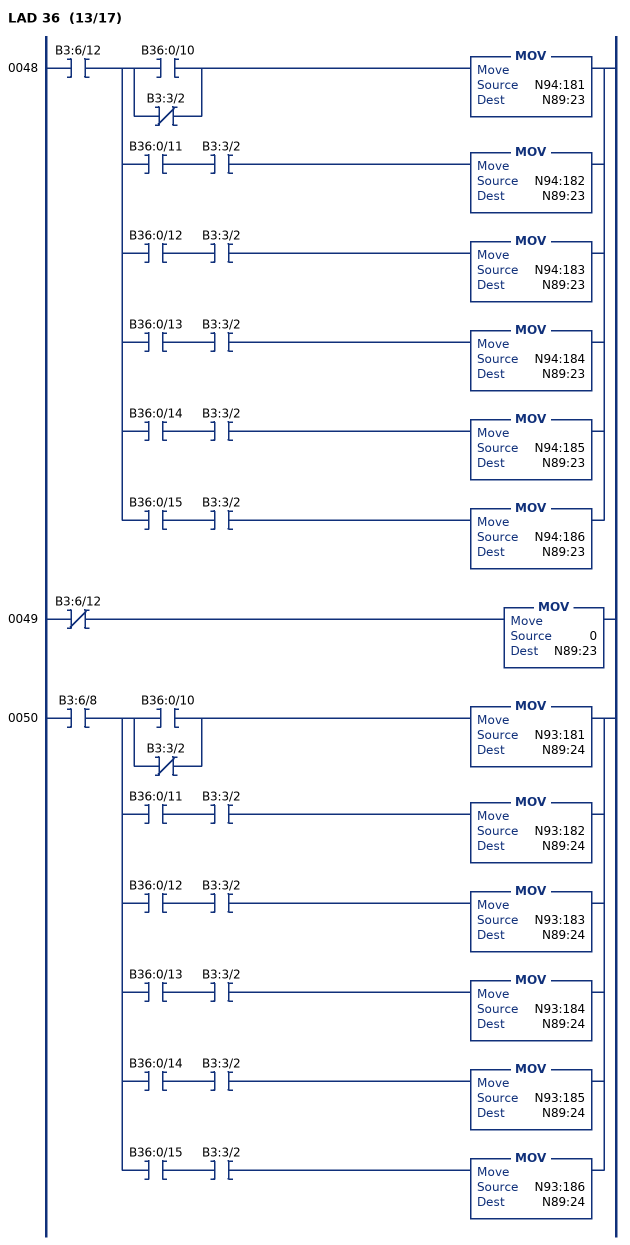
% Rung: 48 %
SOR XIC B3:6/12 BST BST XIC B36:0/10 NXB XIO B3:3/2 BND MOV N94:181 N89:23 NXB XIC B36:0/11 XIC B3:3/2 MOV N94:182 N89:23 NXB XIC B36:0/12 XIC B3:3/2 MOV N94:183 N89:23 NXB XIC B36:0/13 XIC B3:3/2 MOV N94:184 N89:23 NXB XIC B36:0/14 XIC B3:3/2 MOV N94:185 N89:23 NXB XIC B36:0/15 XIC B3:3/2 MOV N94:186 N89:23 BND EOR
% Rung: 49 %
SOR XIO B3:6/12 MOV 0 N89:23 EOR
% Rung: 50 %
SOR XIC B3:6/8 BST BST XIC B36:0/10 NXB XIO B3:3/2 BND MOV N93:181 N89:24 NXB XIC B36:0/11 XIC B3:3/2 MOV N93:182 N89:24 NXB XIC B36:0/12 XIC B3:3/2 MOV N93:183 N89:24 NXB XIC B36:0/13 XIC B3:3/2 MOV N93:184 N89:24 NXB XIC B36:0/14 XIC B3:3/2 MOV N93:185 N89:24 NXB XIC B36:0/15 XIC B3:3/2 MOV N93:186 N89:24 BND EOR

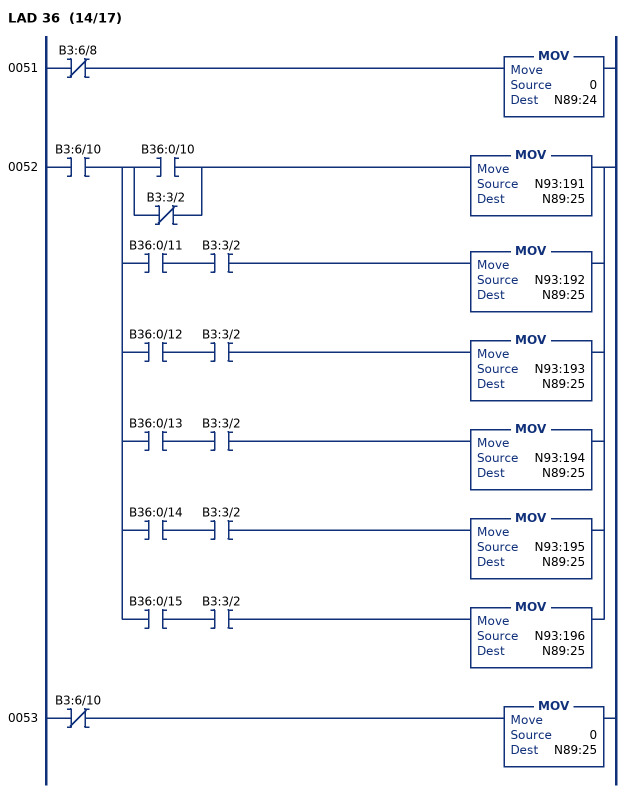
% Rung: 51 %
SOR XIO B3:6/8 MOV 0 N89:24 EOR
% Rung: 52 %
SOR XIC B3:6/10 BST BST XIC B36:0/10 NXB XIO B3:3/2 BND MOV N93:191 N89:25 NXB XIC B36:0/11 XIC B3:3/2 MOV N93:192 N89:25 NXB XIC B36:0/12 XIC B3:3/2 MOV N93:193 N89:25 NXB XIC B36:0/13 XIC B3:3/2 MOV N93:194 N89:25 NXB XIC B36:0/14 XIC B3:3/2 MOV N93:195 N89:25 NXB XIC B36:0/15 XIC B3:3/2 MOV N93:196 N89:25 BND EOR
% Rung: 53 %
SOR XIO B3:6/10 MOV 0 N89:25 EOR

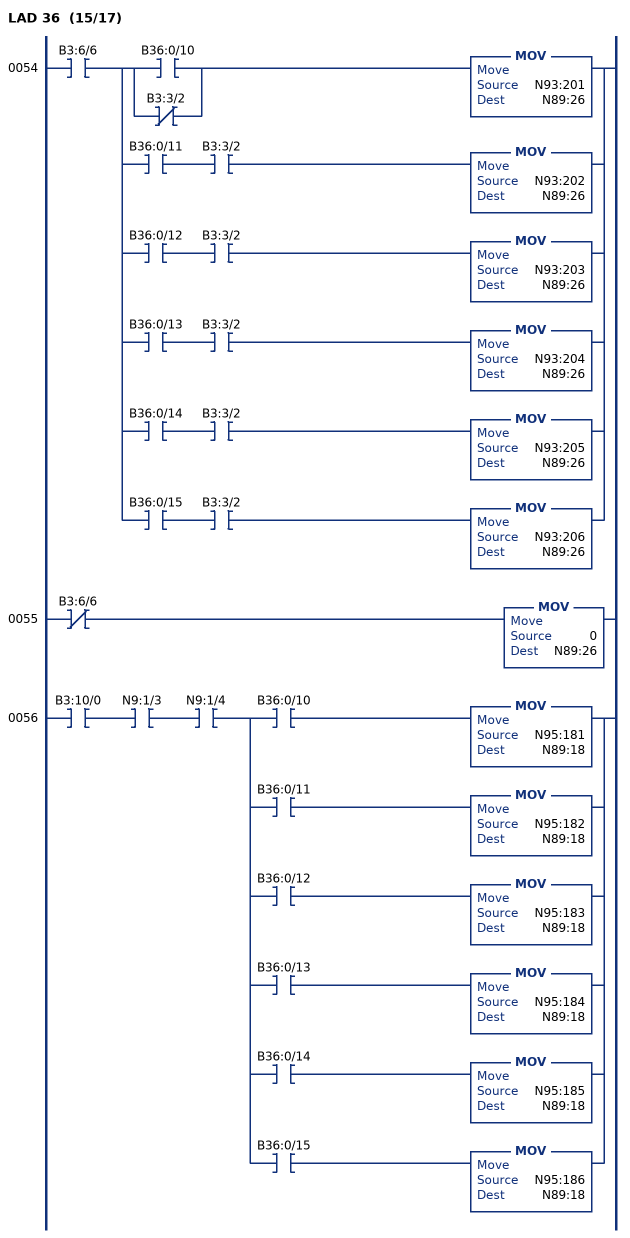
% Rung: 54 %
SOR XIC B3:6/6 BST BST XIC B36:0/10 NXB XIO B3:3/2 BND MOV N93:201 N89:26 NXB XIC B36:0/11 XIC B3:3/2 MOV N93:202 N89:26 NXB XIC B36:0/12 XIC B3:3/2 MOV N93:203 N89:26 NXB XIC B36:0/13 XIC B3:3/2 MOV N93:204 N89:26 NXB XIC B36:0/14 XIC B3:3/2 MOV N93:205 N89:26 NXB XIC B36:0/15 XIC B3:3/2 MOV N93:206 N89:26 BND EOR
% Rung: 55 %
SOR XIO B3:6/6 MOV 0 N89:26 EOR
% Rung: 56 %
SOR XIC B3:10/0 XIC N9:1/3 XIC N9:1/4 BST XIC B36:0/10 MOV N95:181 N89:18 NXB XIC B36:0/11 MOV N95:182 N89:18 NXB XIC B36:0/12 MOV N95:183 N89:18 NXB XIC B36:0/13 MOV N95:184 N89:18 NXB XIC B36:0/14 MOV N95:185 N89:18 NXB XIC B36:0/15 MOV N95:186 N89:18 BND EOR

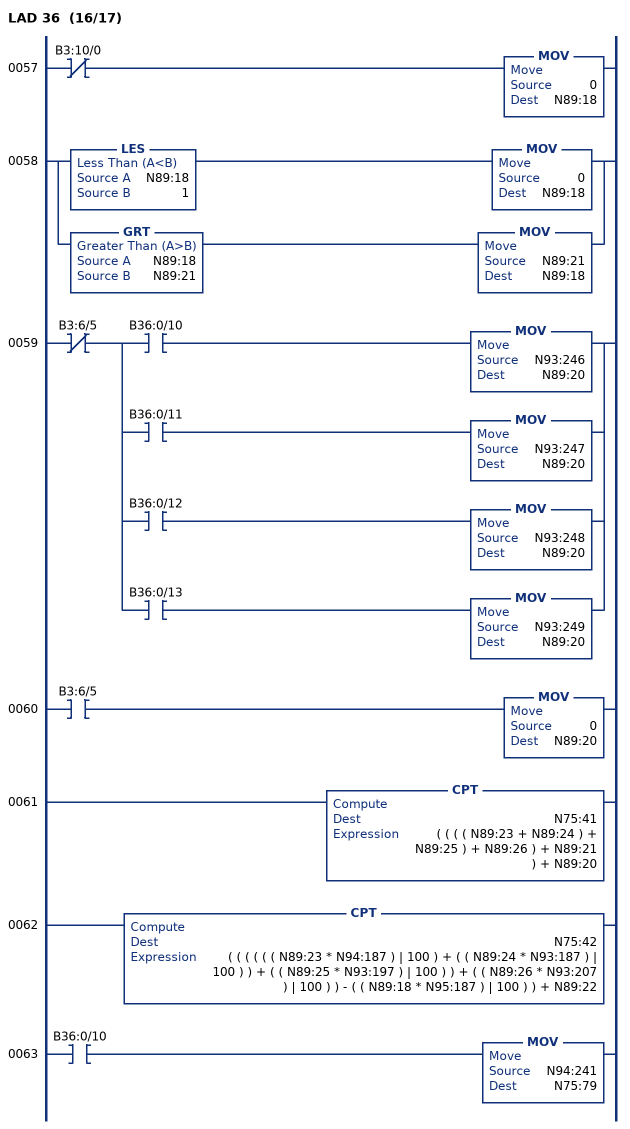
% Rung: 57 %
SOR XIO B3:10/0 MOV 0 N89:18 EOR
% Rung: 58 %
SOR BST LES N89:18 1 MOV 0 N89:18 NXB GRT N89:18 N89:21 MOV N89:21 N89:18 BND EOR
% Rung: 59 %
SOR XIO B3:6/5 BST XIC B36:0/10 MOV N93:246 N89:20 NXB XIC B36:0/11 MOV N93:247 N89:20 NXB XIC B36:0/12 MOV N93:248 N89:20 NXB XIC B36:0/13 MOV N93:249 N89:20 BND EOR
% Rung: 60 %
SOR XIC B3:6/5 MOV 0 N89:20 EOR
% Rung: 61 %
SOR CPT N75:41 " ( ( ( ( N89:23 + N89:24 ) + N89:25 ) + N89:26 ) + N89:21 ) + N89:20 " EOR
% Rung: 62 %
SOR CPT N75:42 " ( ( ( ( ( ( N89:23 * N94:187 ) | 100 ) + ( ( N89:24 * N93:187 ) | 100 ) ) + ( ( N89:25 * N93:197 ) | 100 ) ) + ( ( N89:26 * N93:207 ) | 100 ) ) - ( ( N89:18 * N95:187 ) | 100 ) ) + N89:22 " EOR
% Rung: 63 %
SOR XIC B36:0/10 MOV N94:241 N75:79 EOR

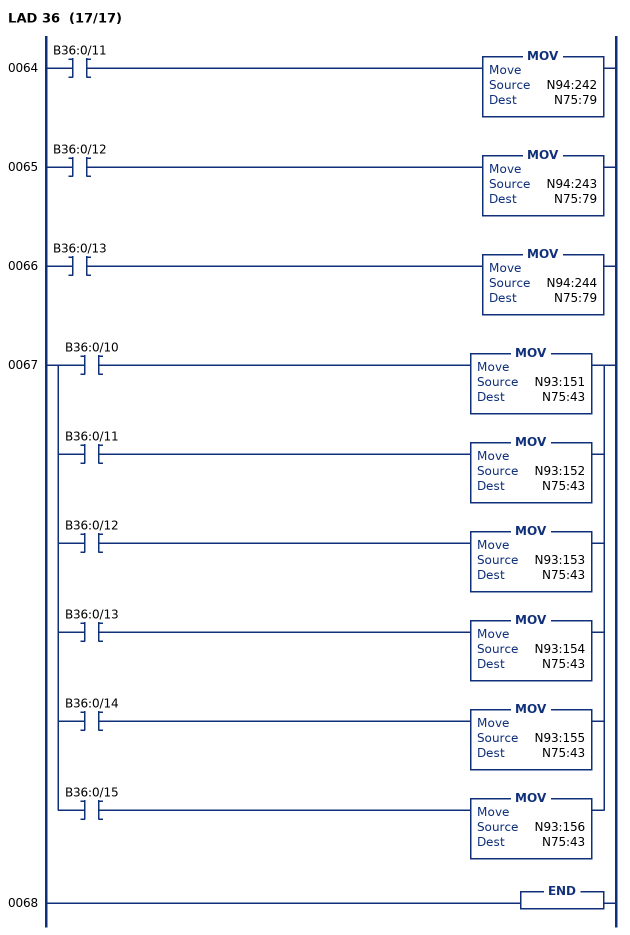
% Rung: 64 %
SOR XIC B36:0/11 MOV N94:242 N75:79 EOR
% Rung: 65 %
SOR XIC B36:0/12 MOV N94:243 N75:79 EOR
% Rung: 66 %
SOR XIC B36:0/13 MOV N94:244 N75:79 EOR
% Rung: 67 %
SOR BST XIC B36:0/10 MOV N93:151 N75:43 NXB XIC B36:0/11 MOV N93:152 N75:43 NXB XIC B36:0/12 MOV N93:153 N75:43 NXB XIC B36:0/13 MOV N93:154 N75:43 NXB XIC B36:0/14 MOV N93:155 N75:43 NXB XIC B36:0/15 MOV N93:156 N75:43 BND EOR
% Rung: 68 %
SOR END EOR

LADDER 41
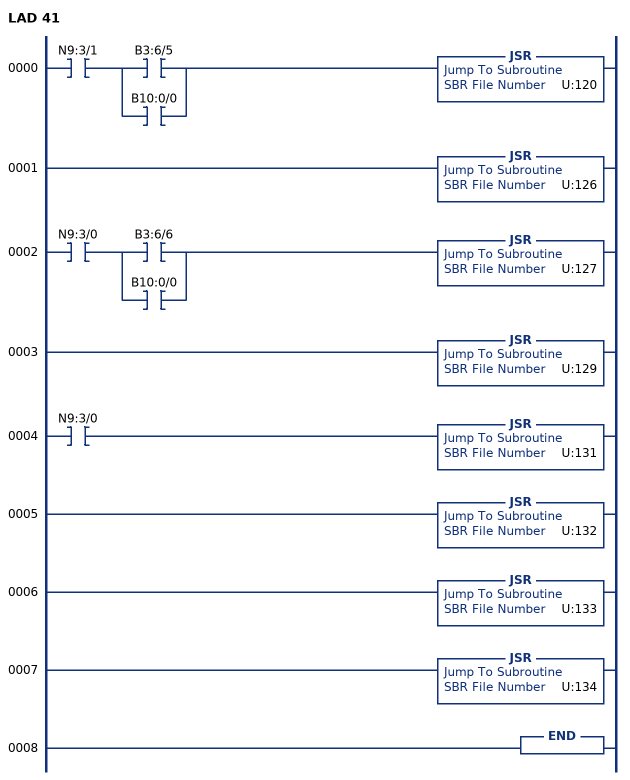
% Rung: 0 %
SOR XIC N9:3/1 BST XIC B3:6/5 NXB XIC B10:0/0 BND JSR U:120 EOR
% Rung: 1 %
SOR JSR U:126 EOR
% Rung: 2 %
SOR XIC N9:3/0 BST XIC B3:6/6 NXB XIC B10:0/0 BND JSR U:127 EOR
% Rung: 3 %
SOR JSR U:129 EOR
% Rung: 4 %
SOR XIC N9:3/0 JSR U:131 EOR
% Rung: 5 %
SOR JSR U:132 EOR
% Rung: 6 %
SOR JSR U:133 EOR
% Rung: 7 %
SOR JSR U:134 EOR
% Rung: 8 %
SOR END EOR

LADDER 50
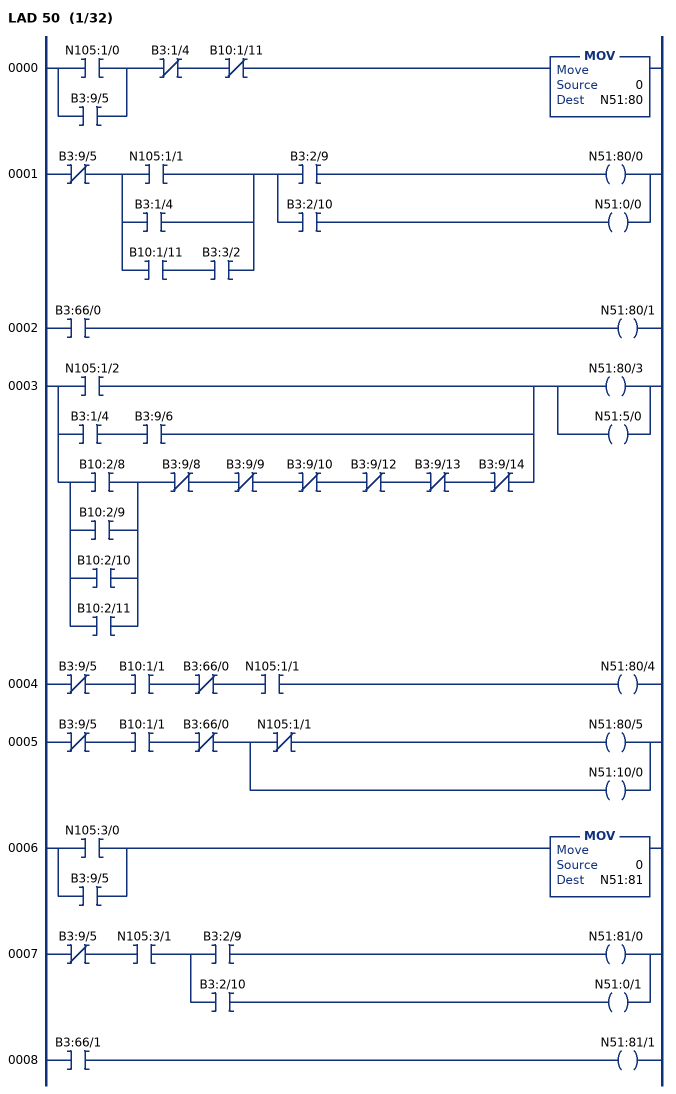
% Rung: 0 %
SOR BST XIC N105:1/0 NXB XIC B3:9/5 BND XIO B3:1/4 XIO B10:1/11 MOV 0 N51:80 EOR
% Rung: 1 %
SOR XIO B3:9/5 BST XIC N105:1/1 NXB XIC B3:1/4 NXB XIC B10:1/11 XIC B3:3/2 BND BST XIC B3:2/9 OTE N51:80/0 NXB XIC B3:2/10 OTE N51:0/0 BND EOR
% Rung: 2 %
SOR XIC B3:66/0 OTE N51:80/1 EOR
% Rung: 3 %
SOR BST XIC N105:1/2 NXB XIC B3:1/4 XIC B3:9/6 NXB BST XIC B10:2/8 NXB XIC B10:2/9 NXB XIC B10:2/10 NXB XIC B10:2/11 BND XIO B3:9/8 XIO B3:9/9 XIO B3:9/10 XIO B3:9/12 XIO B3:9/13 XIO B3:9/14 BND BST OTE N51:80/3 NXB OTE N51:5/0 BND EOR
% Rung: 4 %
SOR XIO B3:9/5 XIC B10:1/1 XIO B3:66/0 XIC N105:1/1 OTE N51:80/4 EOR
% Rung: 5 %
SOR XIO B3:9/5 XIC B10:1/1 XIO B3:66/0 BST XIO N105:1/1 OTE N51:80/5 NXB OTE N51:10/0 BND EOR
% Rung: 6 %
SOR BST XIC N105:3/0 NXB XIC B3:9/5 BND MOV 0 N51:81 EOR
% Rung: 7 %
SOR XIO B3:9/5 XIC N105:3/1 BST XIC B3:2/9 OTE N51:81/0 NXB XIC B3:2/10 OTE N51:0/1 BND EOR
% Rung: 8 %
SOR XIC B3:66/1 OTE N51:81/1 EOR

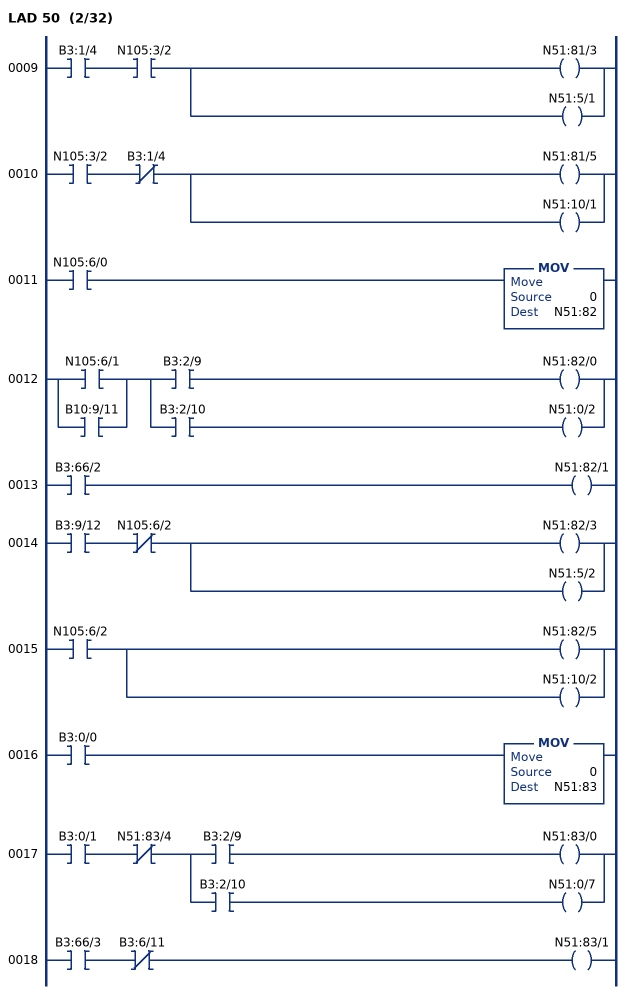
% Rung: 9 %
SOR XIC B3:1/4 XIC N105:3/2 BST OTE N51:81/3 NXB OTE N51:5/1 BND EOR
% Rung: 10 %
SOR XIC N105:3/2 XIO B3:1/4 BST OTE N51:81/5 NXB OTE N51:10/1 BND EOR
% Rung: 11 %
SOR XIC N105:6/0 MOV 0 N51:82 EOR
% Rung: 12 %
SOR BST XIC N105:6/1 NXB XIC B10:9/11 BND BST XIC B3:2/9 OTE N51:82/0 NXB XIC B3:2/10 OTE N51:0/2 BND EOR
% Rung: 13 %
SOR XIC B3:66/2 OTE N51:82/1 EOR
% Rung: 14 %
SOR XIC B3:9/12 XIO N105:6/2 BST OTE N51:82/3 NXB OTE N51:5/2 BND EOR
% Rung: 15 %
SOR XIC N105:6/2 BST OTE N51:82/5 NXB OTE N51:10/2 BND EOR
% Rung: 16 %
SOR XIC B3:0/0 MOV 0 N51:83 EOR
% Rung: 17 %
SOR XIC B3:0/1 XIO N51:83/4 BST XIC B3:2/9 OTE N51:83/0 NXB XIC B3:2/10 OTE N51:0/7 BND EOR
% Rung: 18 %
SOR XIC B3:66/3 XIO B3:6/11 OTE N51:83/1 EOR

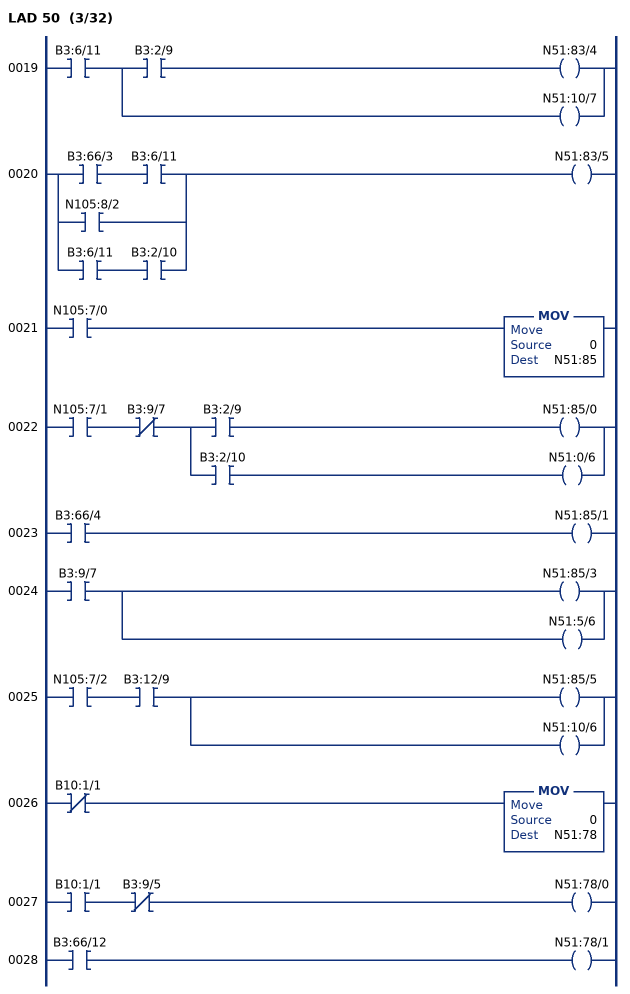
% Rung: 19 %
SOR XIC B3:6/11 BST XIC B3:2/9 OTE N51:83/4 NXB OTE N51:10/7 BND EOR
% Rung: 20 %
SOR BST XIC B3:66/3 XIC B3:6/11 NXB XIC N105:8/2 NXB XIC B3:6/11 XIC B3:2/10 BND OTE N51:83/5 EOR
% Rung: 21 %
SOR XIC N105:7/0 MOV 0 N51:85 EOR
% Rung: 22 %
SOR XIC N105:7/1 XIO B3:9/7 BST XIC B3:2/9 OTE N51:85/0 NXB XIC B3:2/10 OTE N51:0/6 BND EOR
% Rung: 23 %
SOR XIC B3:66/4 OTE N51:85/1 EOR
% Rung: 24 %
SOR XIC B3:9/7 BST OTE N51:85/3 NXB OTE N51:5/6 BND EOR
% Rung: 25 %
SOR XIC N105:7/2 XIC B3:12/9 BST OTE N51:85/5 NXB OTE N51:10/6 BND EOR
% Rung: 26 %
SOR XIO B10:1/1 MOV 0 N51:78 EOR
% Rung: 27 %
SOR XIC B10:1/1 XIO B3:9/5 OTE N51:78/0 EOR
% Rung: 28 %
SOR XIC B3:66/12 OTE N51:78/1 EOR

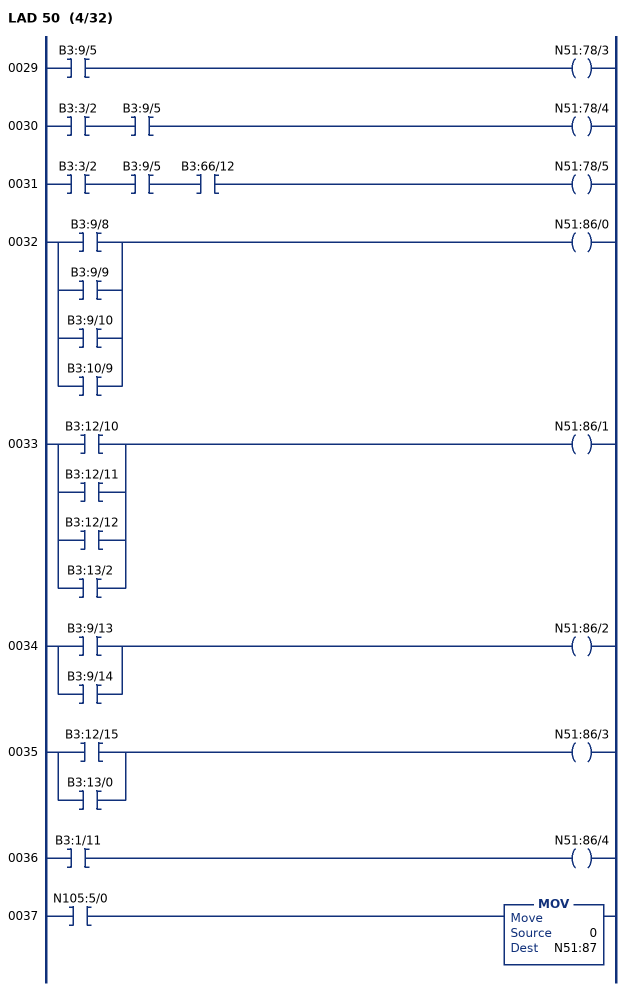
% Rung: 29 %
SOR XIC B3:9/5 OTE N51:78/3 EOR
% Rung: 30 %
SOR XIC B3:3/2 XIC B3:9/5 OTE N51:78/4 EOR
% Rung: 31 %
SOR XIC B3:3/2 XIC B3:9/5 XIC B3:66/12 OTE N51:78/5 EOR
% Rung: 32 %
SOR BST XIC B3:9/8 NXB XIC B3:9/9 NXB XIC B3:9/10 NXB XIC B3:10/9 BND OTE N51:86/0 EOR
% Rung: 33 %
SOR BST XIC B3:12/10 NXB XIC B3:12/11 NXB XIC B3:12/12 NXB XIC B3:13/2 BND OTE N51:86/1 EOR
% Rung: 34 %
SOR BST XIC B3:9/13 NXB XIC B3:9/14 BND OTE N51:86/2 EOR
% Rung: 35 %
SOR BST XIC B3:12/15 NXB XIC B3:13/0 BND OTE N51:86/3 EOR
% Rung: 36 %
SOR XIC B3:1/11 OTE N51:86/4 EOR
% Rung: 37 %
SOR XIC N105:5/0 MOV 0 N51:87 EOR

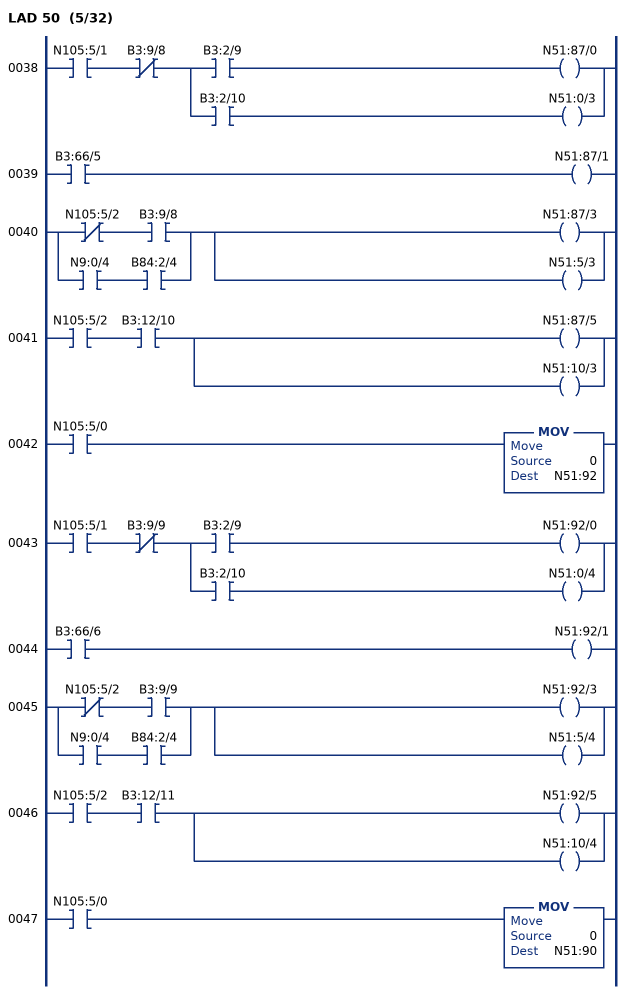
% Rung: 38 %
SOR XIC N105:5/1 XIO B3:9/8 BST XIC B3:2/9 OTE N51:87/0 NXB XIC B3:2/10 OTE N51:0/3 BND EOR
% Rung: 39 %
SOR XIC B3:66/5 OTE N51:87/1 EOR
% Rung: 40 %
SOR BST XIO N105:5/2 XIC B3:9/8 NXB XIC N9:0/4 XIC B84:2/4 BND BST OTE N51:87/3 NXB OTE N51:5/3 BND EOR
% Rung: 41 %
SOR XIC N105:5/2 XIC B3:12/10 BST OTE N51:87/5 NXB OTE N51:10/3 BND EOR
% Rung: 42 %
SOR XIC N105:5/0 MOV 0 N51:92 EOR
% Rung: 43 %
SOR XIC N105:5/1 XIO B3:9/9 BST XIC B3:2/9 OTE N51:92/0 NXB XIC B3:2/10 OTE N51:0/4 BND EOR
% Rung: 44 %
SOR XIC B3:66/6 OTE N51:92/1 EOR
% Rung: 45 %
SOR BST XIO N105:5/2 XIC B3:9/9 NXB XIC N9:0/4 XIC B84:2/4 BND BST OTE N51:92/3 NXB OTE N51:5/4 BND EOR
% Rung: 46 %
SOR XIC N105:5/2 XIC B3:12/11 BST OTE N51:92/5 NXB OTE N51:10/4 BND EOR
% Rung: 47 %
SOR XIC N105:5/0 MOV 0 N51:90 EOR

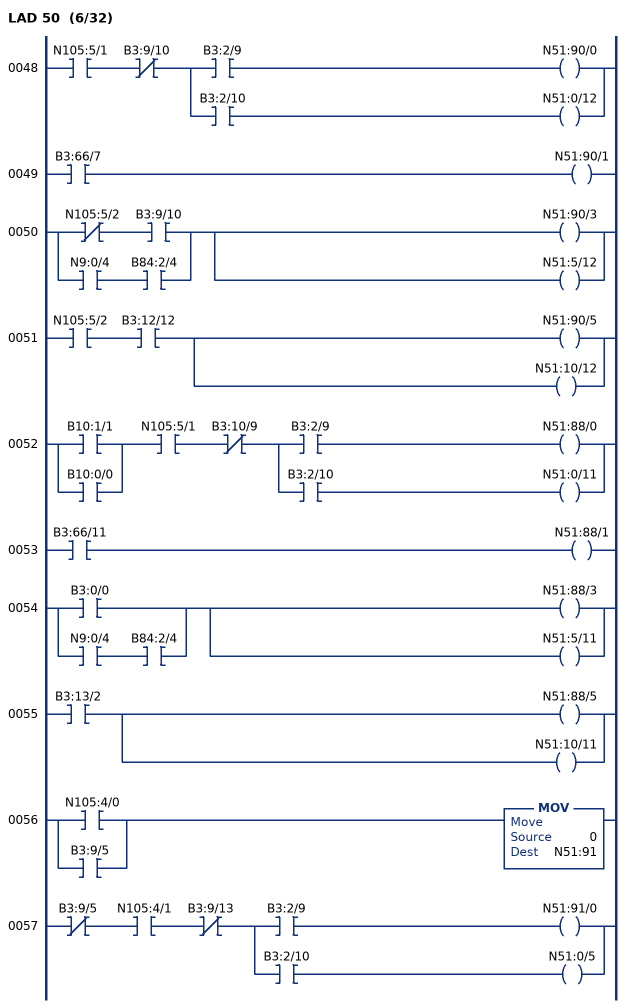
% Rung: 48 %
SOR XIC N105:5/1 XIO B3:9/10 BST XIC B3:2/9 OTE N51:90/0 NXB XIC B3:2/10 OTE N51:0/12 BND EOR
% Rung: 49 %
SOR XIC B3:66/7 OTE N51:90/1 EOR
% Rung: 50 %
SOR BST XIO N105:5/2 XIC B3:9/10 NXB XIC N9:0/4 XIC B84:2/4 BND BST OTE N51:90/3 NXB OTE N51:5/12 BND EOR
% Rung: 51 %
SOR XIC N105:5/2 XIC B3:12/12 BST OTE N51:90/5 NXB OTE N51:10/12 BND EOR
% Rung: 52 %
SOR BST XIC B10:1/1 NXB XIC B10:0/0 BND XIC N105:5/1 XIO B3:10/9 BST XIC B3:2/9 OTE N51:88/0 NXB XIC B3:2/10 OTE N51:0/11 BND EOR
% Rung: 53 %
SOR XIC B3:66/11 OTE N51:88/1 EOR
% Rung: 54 %
SOR BST XIC B3:0/0 NXB XIC N9:0/4 XIC B84:2/4 BND BST OTE N51:88/3 NXB OTE N51:5/11 BND EOR
% Rung: 55 %
SOR XIC B3:13/2 BST OTE N51:88/5 NXB OTE N51:10/11 BND EOR
% Rung: 56 %
SOR BST XIC N105:4/0 NXB XIC B3:9/5 BND MOV 0 N51:91 EOR
% Rung: 57 %
SOR XIO B3:9/5 XIC N105:4/1 XIO B3:9/13 BST XIC B3:2/9 OTE N51:91/0 NXB XIC B3:2/10 OTE N51:0/5 BND EOR

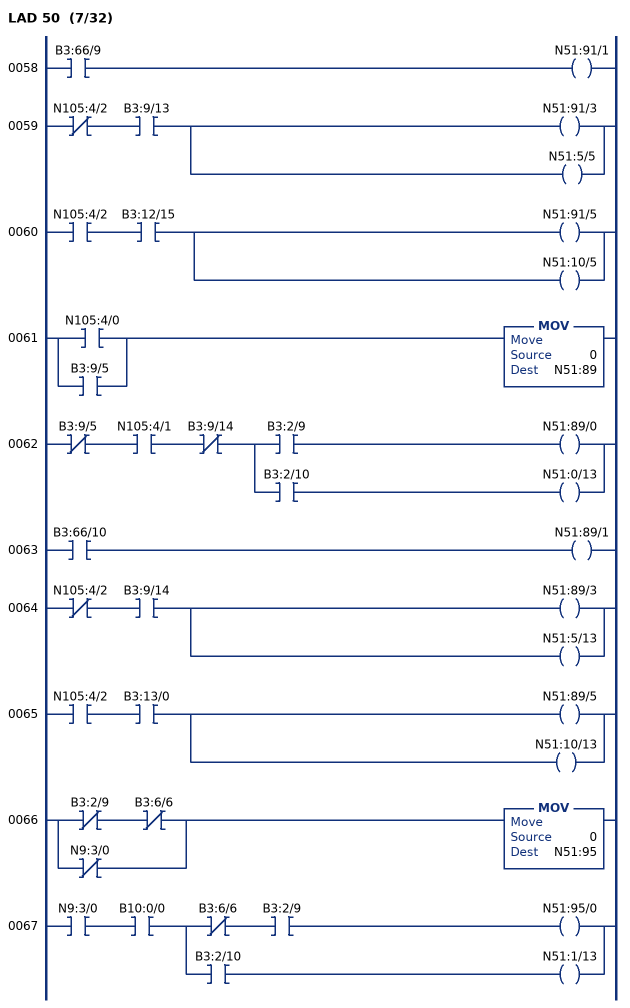
% Rung: 58 %
SOR XIC B3:66/9 OTE N51:91/1 EOR
% Rung: 59 %
SOR XIO N105:4/2 XIC B3:9/13 BST OTE N51:91/3 NXB OTE N51:5/5 BND EOR
% Rung: 60 %
SOR XIC N105:4/2 XIC B3:12/15 BST OTE N51:91/5 NXB OTE N51:10/5 BND EOR
% Rung: 61 %
SOR BST XIC N105:4/0 NXB XIC B3:9/5 BND MOV 0 N51:89 EOR
% Rung: 62 %
SOR XIO B3:9/5 XIC N105:4/1 XIO B3:9/14 BST XIC B3:2/9 OTE N51:89/0 NXB XIC B3:2/10 OTE N51:0/13 BND EOR
% Rung: 63 %
SOR XIC B3:66/10 OTE N51:89/1 EOR
% Rung: 64 %
SOR XIO N105:4/2 XIC B3:9/14 BST OTE N51:89/3 NXB OTE N51:5/13 BND EOR
% Rung: 65 %
SOR XIC N105:4/2 XIC B3:13/0 BST OTE N51:89/5 NXB OTE N51:10/13 BND EOR
% Rung: 66 %
SOR BST XIO B3:2/9 XIO B3:6/6 NXB XIO N9:3/0 BND MOV 0 N51:95 EOR
% Rung: 67 %
SOR XIC N9:3/0 XIC B10:0/0 BST XIO B3:6/6 XIC B3:2/9 OTE N51:95/0 NXB XIC B3:2/10 OTE N51:1/13 BND EOR

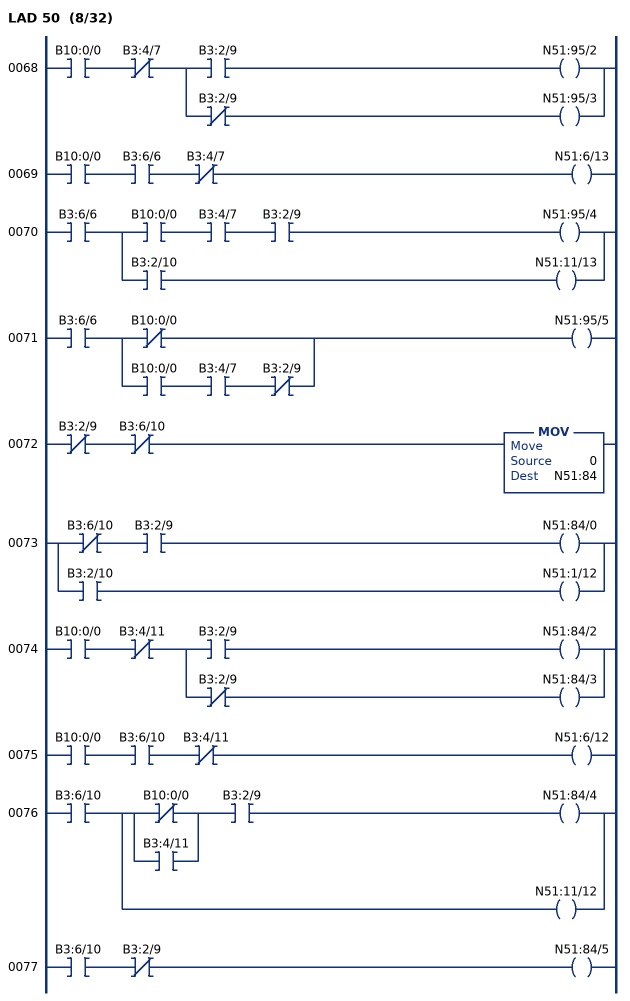
% Rung: 68 %
SOR XIC B10:0/0 XIO B3:4/7 BST XIC B3:2/9 OTE N51:95/2 NXB XIO B3:2/9 OTE N51:95/3 BND EOR
% Rung: 69 %
SOR XIC B10:0/0 XIC B3:6/6 XIO B3:4/7 OTE N51:6/13 EOR
% Rung: 70 %
SOR XIC B3:6/6 BST XIC B10:0/0 XIC B3:4/7 XIC B3:2/9 OTE N51:95/4 NXB XIC B3:2/10 OTE N51:11/13 BND EOR
% Rung: 71 %
SOR XIC B3:6/6 BST XIO B10:0/0 NXB XIC B10:0/0 XIC B3:4/7 XIO B3:2/9 BND OTE N51:95/5 EOR
% Rung: 72 %
SOR XIO B3:2/9 XIO B3:6/10 MOV 0 N51:84 EOR
% Rung: 73 %
SOR BST XIO B3:6/10 XIC B3:2/9 OTE N51:84/0 NXB XIC B3:2/10 OTE N51:1/12 BND EOR
% Rung: 74 %
SOR XIC B10:0/0 XIO B3:4/11 BST XIC B3:2/9 OTE N51:84/2 NXB XIO B3:2/9 OTE N51:84/3 BND EOR
% Rung: 75 %
SOR XIC B10:0/0 XIC B3:6/10 XIO B3:4/11 OTE N51:6/12 EOR
% Rung: 76 %
SOR XIC B3:6/10 BST BST XIO B10:0/0 NXB XIC B3:4/11 BND XIC B3:2/9 OTE N51:84/4 NXB OTE N51:11/12 BND EOR
% Rung: 77 %
SOR XIC B3:6/10 XIO B3:2/9 OTE N51:84/5 EOR

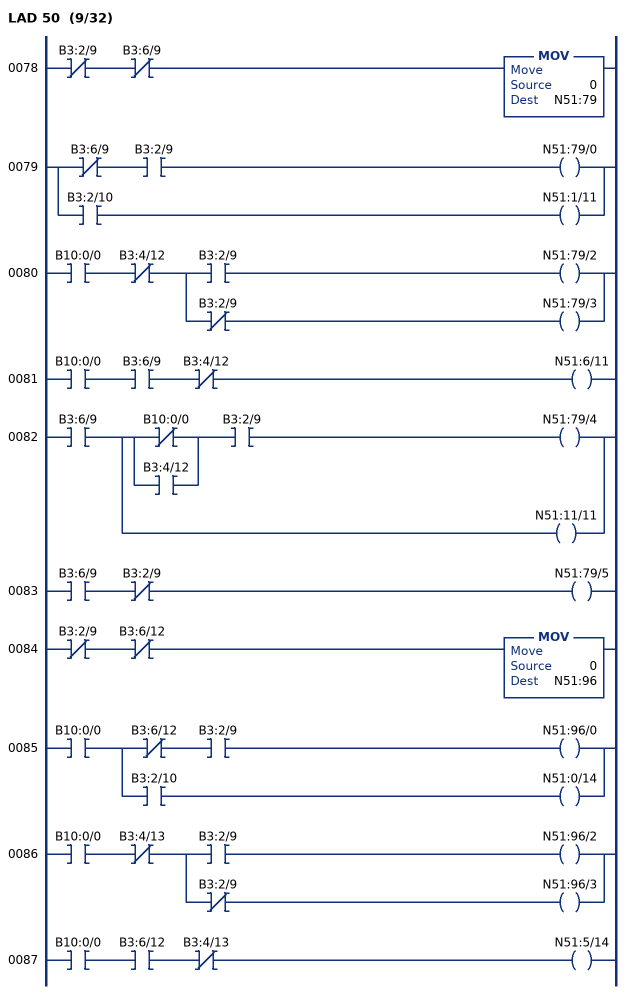
% Rung: 78 %
SOR XIO B3:2/9 XIO B3:6/9 MOV 0 N51:79 EOR
% Rung: 79 %
SOR BST XIO B3:6/9 XIC B3:2/9 OTE N51:79/0 NXB XIC B3:2/10 OTE N51:1/11 BND EOR
% Rung: 80 %
SOR XIC B10:0/0 XIO B3:4/12 BST XIC B3:2/9 OTE N51:79/2 NXB XIO B3:2/9 OTE N51:79/3 BND EOR
% Rung: 81 %
SOR XIC B10:0/0 XIC B3:6/9 XIO B3:4/12 OTE N51:6/11 EOR
% Rung: 82 %
SOR XIC B3:6/9 BST BST XIO B10:0/0 NXB XIC B3:4/12 BND XIC B3:2/9 OTE N51:79/4 NXB OTE N51:11/11 BND EOR
% Rung: 83 %
SOR XIC B3:6/9 XIO B3:2/9 OTE N51:79/5 EOR
% Rung: 84 %
SOR XIO B3:2/9 XIO B3:6/12 MOV 0 N51:96 EOR
% Rung: 85 %
SOR XIC B10:0/0 BST XIO B3:6/12 XIC B3:2/9 OTE N51:96/0 NXB XIC B3:2/10 OTE N51:0/14 BND EOR
% Rung: 86 %
SOR XIC B10:0/0 XIO B3:4/13 BST XIC B3:2/9 OTE N51:96/2 NXB XIO B3:2/9 OTE N51:96/3 BND EOR
% Rung: 87 %
SOR XIC B10:0/0 XIC B3:6/12 XIO B3:4/13 OTE N51:5/14 EOR

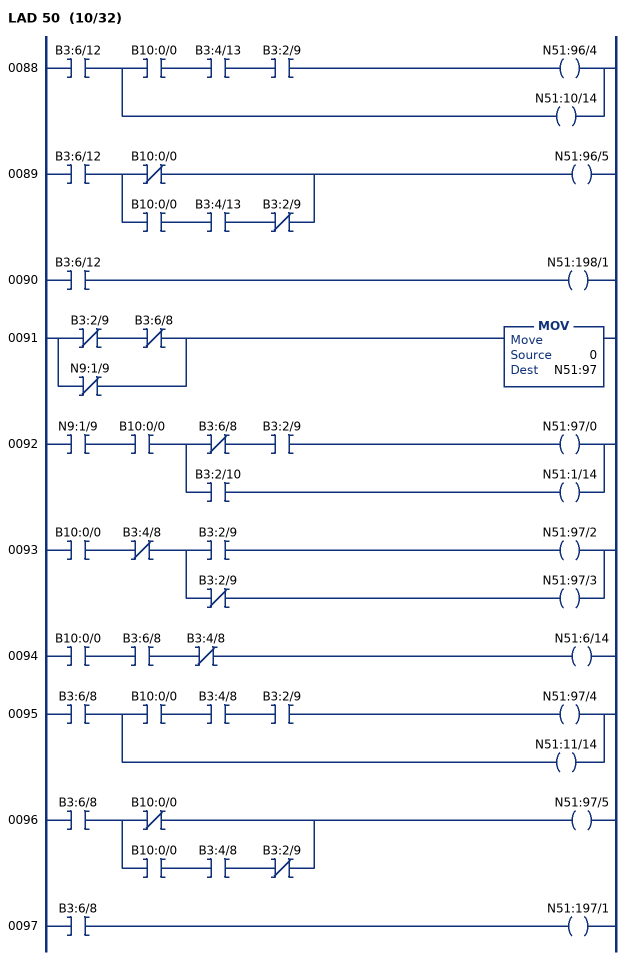
% Rung: 88 %
SOR XIC B3:6/12 BST XIC B10:0/0 XIC B3:4/13 XIC B3:2/9 OTE N51:96/4 NXB OTE N51:10/14 BND EOR
% Rung: 89 %
SOR XIC B3:6/12 BST XIO B10:0/0 NXB XIC B10:0/0 XIC B3:4/13 XIO B3:2/9 BND OTE N51:96/5 EOR
% Rung: 90 %
SOR XIC B3:6/12 OTE N51:198/1 EOR
% Rung: 91 %
SOR BST XIO B3:2/9 XIO B3:6/8 NXB XIO N9:1/9 BND MOV 0 N51:97 EOR
% Rung: 92 %
SOR XIC N9:1/9 XIC B10:0/0 BST XIO B3:6/8 XIC B3:2/9 OTE N51:97/0 NXB XIC B3:2/10 OTE N51:1/14 BND EOR
% Rung: 93 %
SOR XIC B10:0/0 XIO B3:4/8 BST XIC B3:2/9 OTE N51:97/2 NXB XIO B3:2/9 OTE N51:97/3 BND EOR
% Rung: 94 %
SOR XIC B10:0/0 XIC B3:6/8 XIO B3:4/8 OTE N51:6/14 EOR
% Rung: 95 %
SOR XIC B3:6/8 BST XIC B10:0/0 XIC B3:4/8 XIC B3:2/9 OTE N51:97/4 NXB OTE N51:11/14 BND EOR
% Rung: 96 %
SOR XIC B3:6/8 BST XIO B10:0/0 NXB XIC B10:0/0 XIC B3:4/8 XIO B3:2/9 BND OTE N51:97/5 EOR
% Rung: 97 %
SOR XIC B3:6/8 OTE N51:197/1 EOR

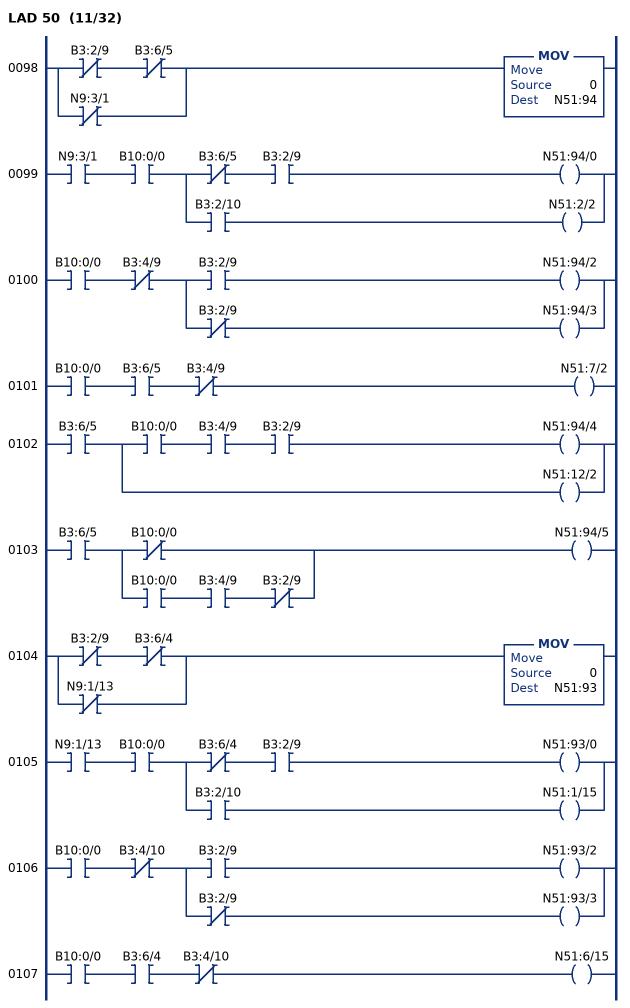
% Rung: 98 %
SOR BST XIO B3:2/9 XIO B3:6/5 NXB XIO N9:3/1 BND MOV 0 N51:94 EOR
% Rung: 99 %
SOR XIC N9:3/1 XIC B10:0/0 BST XIO B3:6/5 XIC B3:2/9 OTE N51:94/0 NXB XIC B3:2/10 OTE N51:2/2 BND EOR
% Rung: 100 %
SOR XIC B10:0/0 XIO B3:4/9 BST XIC B3:2/9 OTE N51:94/2 NXB XIO B3:2/9 OTE N51:94/3 BND EOR
% Rung: 101 %
SOR XIC B10:0/0 XIC B3:6/5 XIO B3:4/9 OTE N51:7/2 EOR
% Rung: 102 %
SOR XIC B3:6/5 BST XIC B10:0/0 XIC B3:4/9 XIC B3:2/9 OTE N51:94/4 NXB OTE N51:12/2 BND EOR
% Rung: 103 %
SOR XIC B3:6/5 BST XIO B10:0/0 NXB XIC B10:0/0 XIC B3:4/9 XIO B3:2/9 BND OTE N51:94/5 EOR
% Rung: 104 %
SOR BST XIO B3:2/9 XIO B3:6/4 NXB XIO N9:1/13 BND MOV 0 N51:93 EOR
% Rung: 105 %
SOR XIC N9:1/13 XIC B10:0/0 BST XIO B3:6/4 XIC B3:2/9 OTE N51:93/0 NXB XIC B3:2/10 OTE N51:1/15 BND EOR
% Rung: 106 %
SOR XIC B10:0/0 XIO B3:4/10 BST XIC B3:2/9 OTE N51:93/2 NXB XIO B3:2/9 OTE N51:93/3 BND EOR
% Rung: 107 %
SOR XIC B10:0/0 XIC B3:6/4 XIO B3:4/10 OTE N51:6/15 EOR

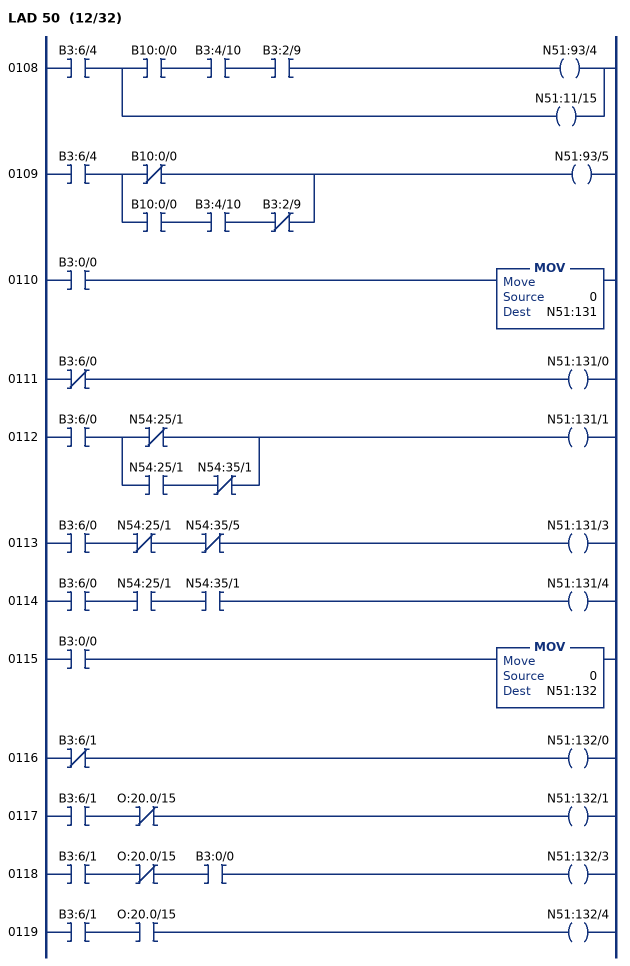
% Rung: 108 %
SOR XIC B3:6/4 BST XIC B10:0/0 XIC B3:4/10 XIC B3:2/9 OTE N51:93/4 NXB OTE N51:11/15 BND EOR
% Rung: 109 %
SOR XIC B3:6/4 BST XIO B10:0/0 NXB XIC B10:0/0 XIC B3:4/10 XIO B3:2/9 BND OTE N51:93/5 EOR
% Rung: 110 %
SOR XIC B3:0/0 MOV 0 N51:131 EOR
% Rung: 111 %
SOR XIO B3:6/0 OTE N51:131/0 EOR
% Rung: 112 %
SOR XIC B3:6/0 BST XIO N54:25/1 NXB XIC N54:25/1 XIO N54:35/1 BND OTE N51:131/1 EOR
% Rung: 113 %
SOR XIC B3:6/0 XIO N54:25/1 XIO N54:35/5 OTE N51:131/3 EOR
% Rung: 114 %
SOR XIC B3:6/0 XIC N54:25/1 XIC N54:35/1 OTE N51:131/4 EOR
% Rung: 115 %
SOR XIC B3:0/0 MOV 0 N51:132 EOR
% Rung: 116 %
SOR XIO B3:6/1 OTE N51:132/0 EOR
% Rung: 117 %
SOR XIC B3:6/1 XIO O:20.0/15 OTE N51:132/1 EOR
% Rung: 118 %
SOR XIC B3:6/1 XIO O:20.0/15 XIC B3:0/0 OTE N51:132/3 EOR
% Rung: 119 %
SOR XIC B3:6/1 XIC O:20.0/15 OTE N51:132/4 EOR

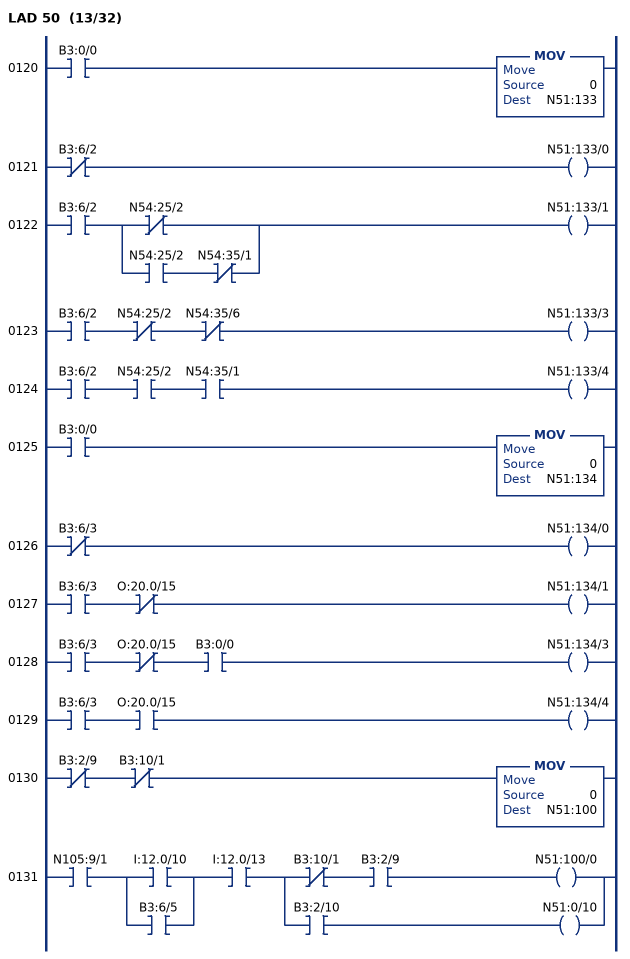
% Rung: 120 %
SOR XIC B3:0/0 MOV 0 N51:133 EOR
% Rung: 121 %
SOR XIO B3:6/2 OTE N51:133/0 EOR
% Rung: 122 %
SOR XIC B3:6/2 BST XIO N54:25/2 NXB XIC N54:25/2 XIO N54:35/1 BND OTE N51:133/1 EOR
% Rung: 123 %
SOR XIC B3:6/2 XIO N54:25/2 XIO N54:35/6 OTE N51:133/3 EOR
% Rung: 124 %
SOR XIC B3:6/2 XIC N54:25/2 XIC N54:35/1 OTE N51:133/4 EOR
% Rung: 125 %
SOR XIC B3:0/0 MOV 0 N51:134 EOR
% Rung: 126 %
SOR XIO B3:6/3 OTE N51:134/0 EOR
% Rung: 127 %
SOR XIC B3:6/3 XIO O:20.0/15 OTE N51:134/1 EOR
% Rung: 128 %
SOR XIC B3:6/3 XIO O:20.0/15 XIC B3:0/0 OTE N51:134/3 EOR
% Rung: 129 %
SOR XIC B3:6/3 XIC O:20.0/15 OTE N51:134/4 EOR
% Rung: 130 %
SOR XIO B3:2/9 XIO B3:10/1 MOV 0 N51:100 EOR
% Rung: 131 %
SOR XIC N105:9/1 BST XIC I:12.0/10 NXB XIC B3:6/5 BND XIC I:12.0/13 BST XIO B3:10/1 XIC B3:2/9 OTE N51:100/0 NXB XIC B3:2/10 OTE N51:0/10 BND EOR

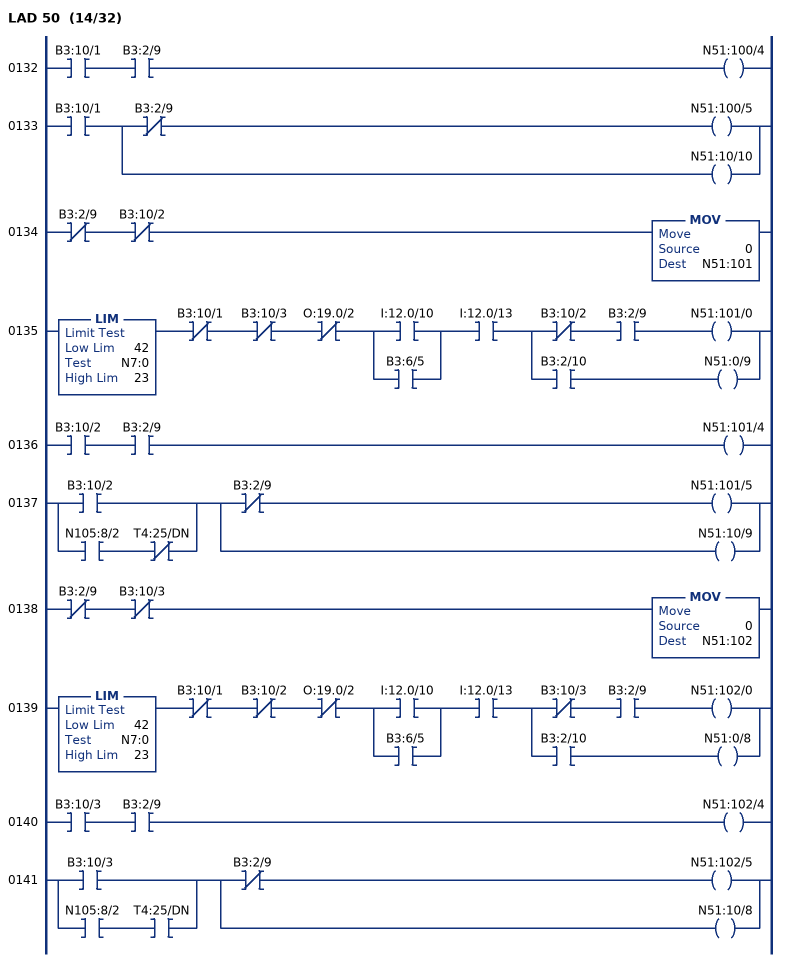
% Rung: 132 %
SOR XIC B3:10/1 XIC B3:2/9 OTE N51:100/4 EOR
% Rung: 133 %
SOR XIC B3:10/1 BST XIO B3:2/9 OTE N51:100/5 NXB OTE N51:10/10 BND EOR
% Rung: 134 %
SOR XIO B3:2/9 XIO B3:10/2 MOV 0 N51:101 EOR
% Rung: 135 %
SOR LIM 42 N7:0 23 XIO B3:10/1 XIO B3:10/3 XIO O:19.0/2 BST XIC I:12.0/10 NXB XIC B3:6/5 BND XIC I:12.0/13 BST XIO B3:10/2 XIC B3:2/9 OTE N51:101/0 NXB XIC B3:2/10 OTE N51:0/9 BND EOR
% Rung: 136 %
SOR XIC B3:10/2 XIC B3:2/9 OTE N51:101/4 EOR
% Rung: 137 %
SOR BST XIC B3:10/2 NXB XIC N105:8/2 XIO T4:25/DN BND BST XIO B3:2/9 OTE N51:101/5 NXB OTE N51:10/9 BND EOR
% Rung: 138 %
SOR XIO B3:2/9 XIO B3:10/3 MOV 0 N51:102 EOR
% Rung: 139 %
SOR LIM 42 N7:0 23 XIO B3:10/1 XIO B3:10/2 XIO O:19.0/2 BST XIC I:12.0/10 NXB XIC B3:6/5 BND XIC I:12.0/13 BST XIO B3:10/3 XIC B3:2/9 OTE N51:102/0 NXB XIC B3:2/10 OTE N51:0/8 BND EOR
% Rung: 140 %
SOR XIC B3:10/3 XIC B3:2/9 OTE N51:102/4 EOR
% Rung: 141 %
SOR BST XIC B3:10/3 NXB XIC N105:8/2 XIC T4:25/DN BND BST XIO B3:2/9 OTE N51:102/5 NXB OTE N51:10/8 BND EOR

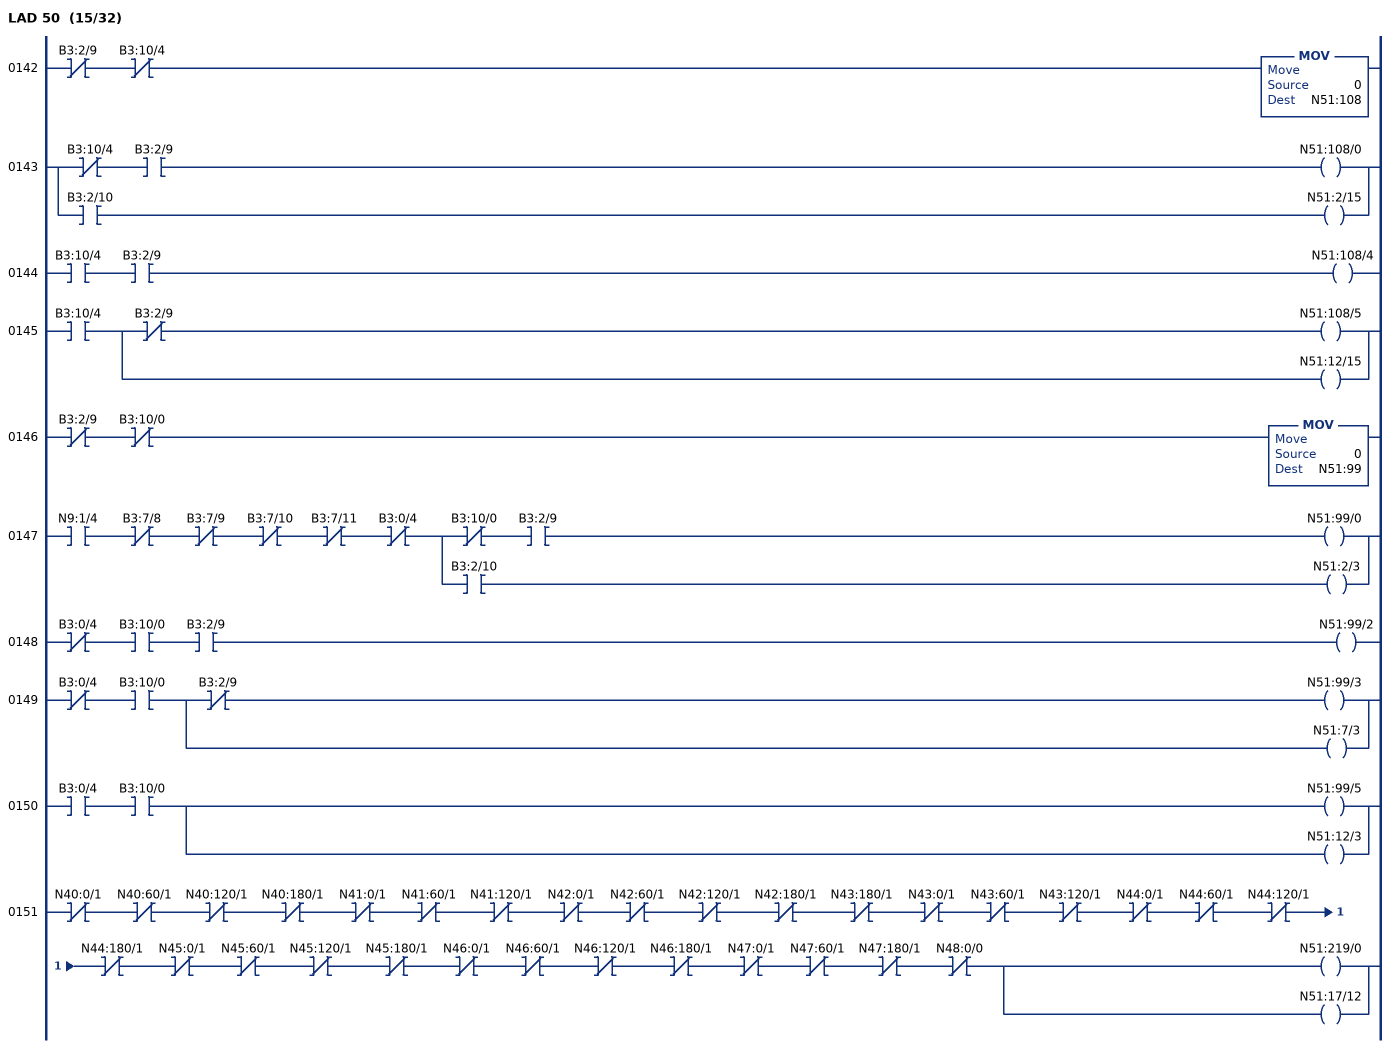
% Rung: 142 %
SOR XIO B3:2/9 XIO B3:10/4 MOV 0 N51:108 EOR
% Rung: 143 %
SOR BST XIO B3:10/4 XIC B3:2/9 OTE N51:108/0 NXB XIC B3:2/10 OTE N51:2/15 BND EOR
% Rung: 144 %
SOR XIC B3:10/4 XIC B3:2/9 OTE N51:108/4 EOR
% Rung: 145 %
SOR XIC B3:10/4 BST XIO B3:2/9 OTE N51:108/5 NXB OTE N51:12/15 BND EOR
% Rung: 146 %
SOR XIO B3:2/9 XIO B3:10/0 MOV 0 N51:99 EOR
% Rung: 147 %
SOR XIC N9:1/4 XIO B3:7/8 XIO B3:7/9 XIO B3:7/10 XIO B3:7/11 XIO B3:0/4 BST XIO B3:10/0 XIC B3:2/9 OTE N51:99/0 NXB XIC B3:2/10 OTE N51:2/3 BND EOR
% Rung: 148 %
SOR XIO B3:0/4 XIC B3:10/0 XIC B3:2/9 OTE N51:99/2 EOR
% Rung: 149 %
SOR XIO B3:0/4 XIC B3:10/0 BST XIO B3:2/9 OTE N51:99/3 NXB OTE N51:7/3 BND EOR
% Rung: 150 %
SOR XIC B3:0/4 XIC B3:10/0 BST OTE N51:99/5 NXB OTE N51:12/3 BND EOR
% Rung: 151 %
SOR XIO N40:0/1 XIO N40:60/1 XIO N40:120/1 XIO N40:180/1 XIO N41:0/1 XIO N41:60/1 XIO N41:120/1 XIO N42:0/1 XIO N42:60/1 XIO N42:120/1 XIO N42:180/1 XIO N43:180/1 XIO N43:0/1 XIO N43:60/1 XIO N43:120/1 XIO N44:0/1 XIO N44:60/1 XIO N44:120/1 XIO N44:180/1 XIO N45:0/1 XIO N45:60/1 XIO N45:120/1 XIO N45:180/1 XIO N46:0/1 XIO N46:60/1 XIO N46:120/1 XIO N46:180/1 XIO N47:0/1 XIO N47:60/1 XIO N47:180/1 XIO N48:0/0 BST OTE N51:219/0 NXB OTE N51:17/12 BND EOR

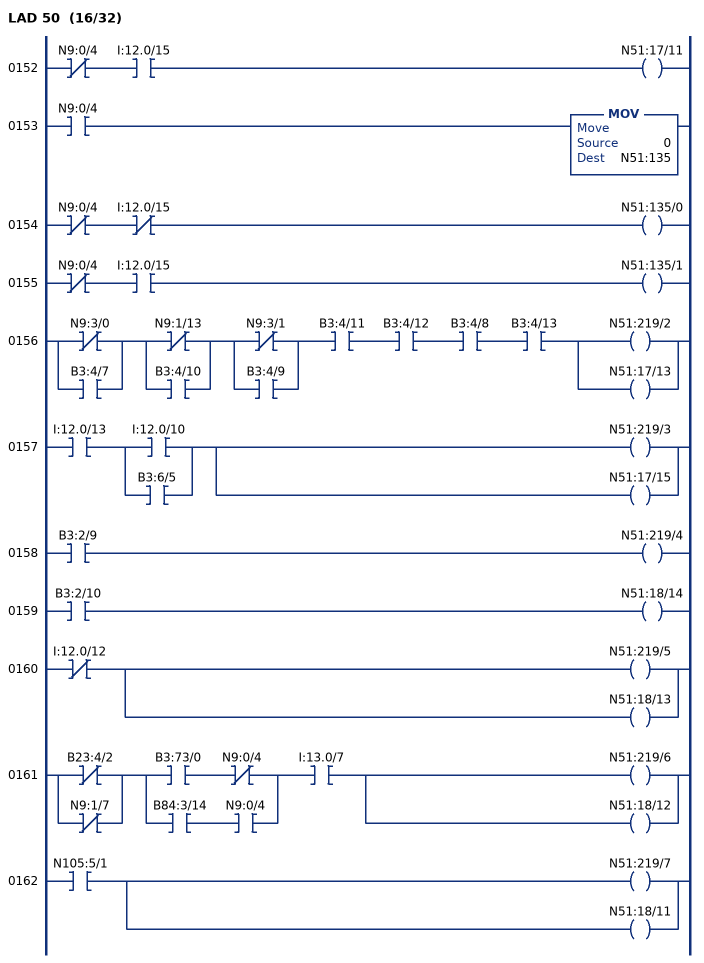
% Rung: 152 %
SOR XIO N9:0/4 XIC I:12.0/15 OTE N51:17/11 EOR
% Rung: 153 %
SOR XIC N9:0/4 MOV 0 N51:135 EOR
% Rung: 154 %
SOR XIO N9:0/4 XIO I:12.0/15 OTE N51:135/0 EOR
% Rung: 155 %
SOR XIO N9:0/4 XIC I:12.0/15 OTE N51:135/1 EOR
% Rung: 156 %
SOR BST XIO N9:3/0 NXB XIC B3:4/7 BND BST XIO N9:1/13 NXB XIC B3:4/10 BND BST XIO N9:3/1 NXB XIC B3:4/9 BND XIC B3:4/11 XIC B3:4/12 XIC B3:4/8 XIC B3:4/13 BST OTE N51:219/2 NXB OTE N51:17/13 BND EOR
% Rung: 157 %
SOR XIC I:12.0/13 BST XIC I:12.0/10 NXB XIC B3:6/5 BND BST OTE N51:219/3 NXB OTE N51:17/15 BND EOR
% Rung: 158 %
SOR XIC B3:2/9 OTE N51:219/4 EOR
% Rung: 159 %
SOR XIC B3:2/10 OTE N51:18/14 EOR
% Rung: 160 %
SOR XIO I:12.0/12 BST OTE N51:219/5 NXB OTE N51:18/13 BND EOR
% Rung: 161 %
SOR BST XIO B23:4/2 NXB XIO N9:1/7 BND BST XIC B3:73/0 XIO N9:0/4 NXB XIC B84:3/14 XIC N9:0/4 BND XIC I:13.0/7 BST OTE N51:219/6 NXB OTE N51:18/12 BND EOR
% Rung: 162 %
SOR XIC N105:5/1 BST OTE N51:219/7 NXB OTE N51:18/11 BND EOR

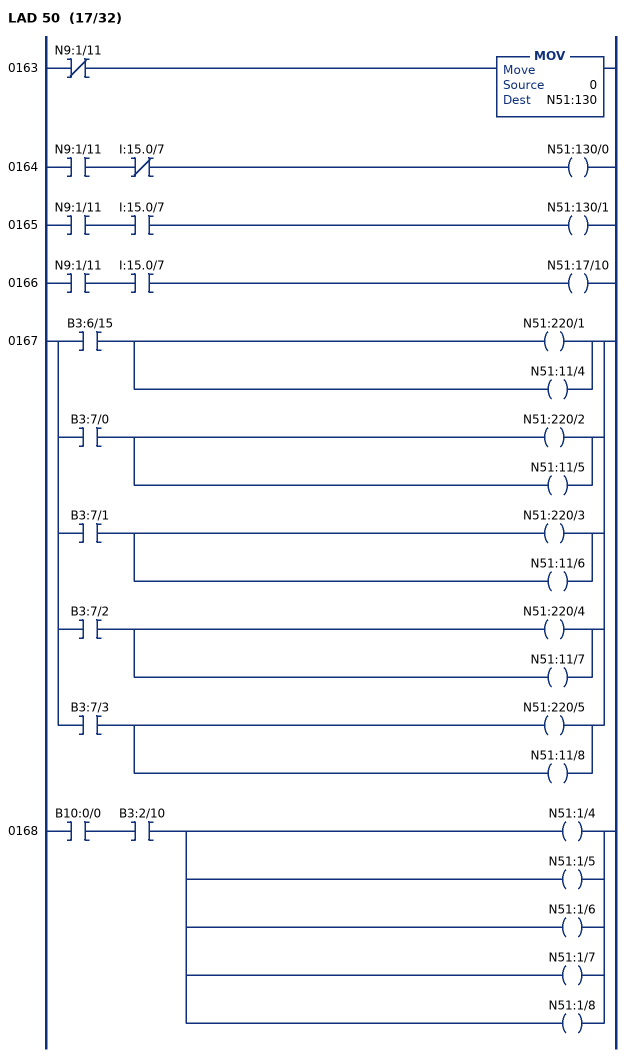
% Rung: 163 %
SOR XIO N9:1/11 MOV 0 N51:130 EOR
% Rung: 164 %
SOR XIC N9:1/11 XIO I:15.0/7 OTE N51:130/0 EOR
% Rung: 165 %
SOR XIC N9:1/11 XIC I:15.0/7 OTE N51:130/1 EOR
% Rung: 166 %
SOR XIC N9:1/11 XIC I:15.0/7 OTE N51:17/10 EOR
% Rung: 167 %
SOR BST XIC B3:6/15 BST OTE N51:220/1 NXB OTE N51:11/4 BND NXB XIC B3:7/0 BST OTE N51:220/2 NXB OTE N51:11/5 BND NXB XIC B3:7/1 BST OTE N51:220/3 NXB OTE N51:11/6 BND NXB XIC B3:7/2 BST OTE N51:220/4 NXB OTE N51:11/7 BND NXB XIC B3:7/3 BST OTE N51:220/5 NXB OTE N51:11/8 BND BND EOR
% Rung: 168 %
SOR XIC B10:0/0 XIC B3:2/10 BST OTE N51:1/4 NXB OTE N51:1/5 NXB OTE N51:1/6 NXB OTE N51:1/7 NXB OTE N51:1/8 BND EOR

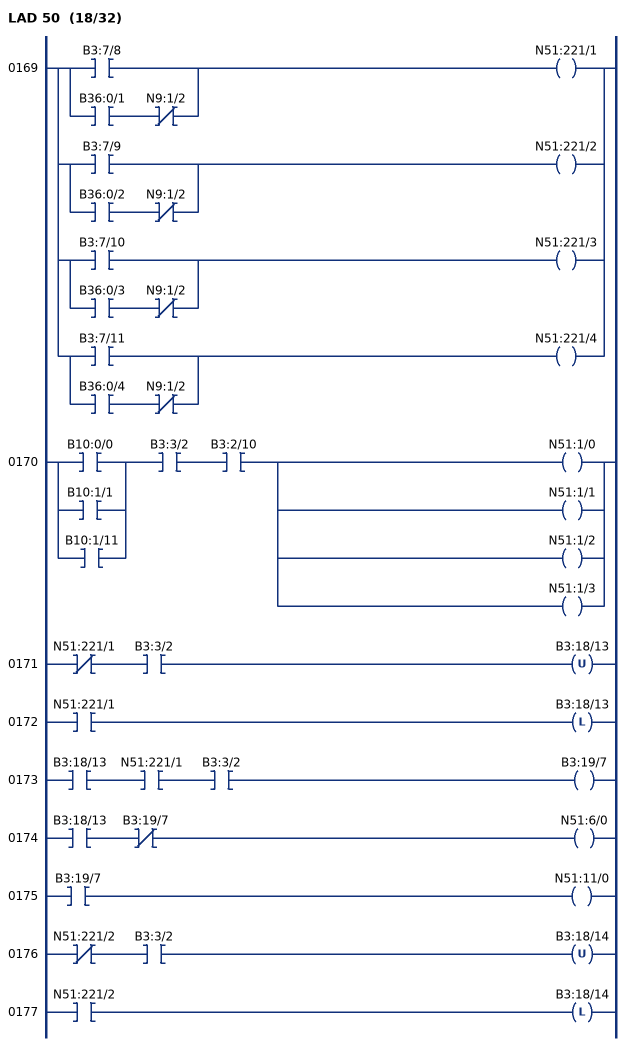
% Rung: 169 %
SOR BST BST XIC B3:7/8 NXB XIC B36:0/1 XIO N9:1/2 BND OTE N51:221/1 NXB BST XIC B3:7/9 NXB XIC B36:0/2 XIO N9:1/2 BND OTE N51:221/2 NXB BST XIC B3:7/10 NXB XIC B36:0/3 XIO N9:1/2 BND OTE N51:221/3 NXB BST XIC B3:7/11 NXB XIC B36:0/4 XIO N9:1/2 BND OTE N51:221/4 BND EOR
% Rung: 170 %
SOR BST XIC B10:0/0 NXB XIC B10:1/1 NXB XIC B10:1/11 BND XIC B3:3/2 XIC B3:2/10 BST OTE N51:1/0 NXB OTE N51:1/1 NXB OTE N51:1/2 NXB OTE N51:1/3 BND EOR
% Rung: 171 %
SOR XIO N51:221/1 XIC B3:3/2 OTU B3:18/13 EOR
% Rung: 172 %
SOR XIC N51:221/1 OTL B3:18/13 EOR
% Rung: 173 %
SOR XIC B3:18/13 XIC N51:221/1 XIC B3:3/2 OTE B3:19/7 EOR
% Rung: 174 %
SOR XIC B3:18/13 XIO B3:19/7 OTE N51:6/0 EOR
% Rung: 175 %
SOR XIC B3:19/7 OTE N51:11/0 EOR
% Rung: 176 %
SOR XIO N51:221/2 XIC B3:3/2 OTU B3:18/14 EOR
% Rung: 177 %
SOR XIC N51:221/2 OTL B3:18/14 EOR

